(* IEC 61131-3 sources: Lasal/CPU_5344_V01/Class/SdiasManager (part 3) *)

            aProperties[1].udPropertyId     := SDM_PROP_BITMAP_APPLICATION_LED_16_31;
            aProperties[1].udPropertyValue  := AppliLEDStates[4]$UDINT;

            aProperties[2].udPropertyId     := SDM_PROP_BITMAP_APPLICATION_LED_32_47;
            aProperties[2].udPropertyValue  := AppliLEDStates[8]$UDINT;

            aProperties[3].udPropertyId     := SDM_PROP_BITMAP_APPLICATION_LED_48_63;
            aProperties[3].udPropertyValue  := AppliLEDStates[12]$UDINT;

            if SDIAS_iSetNodeProperties(hNodeHandle         := udNodeHandle
                                      , udPropertyCount     := 4
                                      , psPropertyValuePairs:= #aProperties[0]
                                      ) <> SDIAS_OK then
#ifdef HWC_LogError
              HWC_LogError(this, "@0067 (SdiasManager::CyWork) Failed to set the application LED states via OS interface!");
#endif
              ErrorInitStep := InitSSW;
              InitSSW := _PrepareError;
              ClassState := _ManagerError;
            else
              b_NewLEDStates := FALSE;
            end_if;
          end_if;
        end_if;
      elsif AsyWriteUsage = _UsedByLED then
        b_NewLEDStates := FALSE;
        AsyWriteUsage := _NotUsed;
      end_if;
    elsif (b_PostInitFinished = FALSE) & InitStartTime & ((ops.tAbsolute - InitStartTime) > (SDIAS_INIT_BLOCK_TIMEOUT + AdditionalPostInitTime)) then
      // timeout for last init if we're stuck in a step for too long (1min). otherwise the plc would not start up, which makes it hard to show the error
#ifdef HWC_LogValue1
      HWC_LogValue1(this, "@0068 (SdiasManager::CyWork) Init has been blocked for too long! Initialisation of SDIAS Manager timed out! Blocked step: 0x{0}",InitSSW$UDINT);
#endif
      ClassState := _TimeoutInInit;
      ErrorInitStep := InitSSW;
      InitSSW := _PrepareError;
    end_if;

  elsif b_PostInitFinished = FALSE then
    // if the module is not online => tell the manager that we're finished with initializing
    SendPostInitFinished(DisableThisObject:=TRUE);

    // set required error, if there is a required module
    SetRequiredError();
  end_if;

  PostRtMessages();

	state := READY;

END_FUNCTION

FUNCTION VIRTUAL GLOBAL SdiasManager::RtWork
	VAR_INPUT
		EAX 	: UDINT;
	END_VAR
	VAR_OUTPUT
		state (EAX) 	: UDINT;
	END_VAR
  VAR
  	calloption          : UDINT;
    i                   : UDINT;
    pModuleInfo         : ^t_ModuleObjectInfo;
    dataSETRUNSTATE     : t_SetRunStateCfg;
    dataResetDO         : t_ResetDOCfg;
    dataSyncData        : t_SyncData;
  	tempCmd             : CmdStruct;
    _result             : results;
    pHelpAccess         : ^t_AccessElement;
    CheckRetryCounters  : BOOL;
    ActFrameCounter     : UDINT;
    TempControlByte     : t_SDIAS_ControlByte;
    dataUPDATEDO        : t_UpdateDOCfg;
    aProperties         : ARRAY [0..4] OF SDM_PROPERTY_VALUE_PAIR;
    SyncInjectionCfg    : t_SyncInjectionCfg;
    CrashThisTime       : USINT;
    aCrashMessage       : ARRAY [0..255] OF CHAR;
    TmpRetryCount       : UDINT;
    TempUDINT           : UDINT;
    ret_code 	          : iprStates;

#ifdef SDIAS_RT_TIME_MEASUREMENT
    Time1           : UDINT;
    Time2           : UDINT;
    TimeTotal1      : UDINT;
    TimeTotal2      : UDINT;
#endif
  END_VAR

  // Called from BusInterface on UpdateRt or UpdateRtPostScan

  // Save state
  // This must be the 1. line in this function or EAX may be overwriten by the generated AWL code
  calloption := EAX;

  if Online then
    pModuleInfo := #ModuleObjInfo[0];
    case RtSSW of
//**********************************************************************************************************************************************************
      _RtIdle: // nothing

//**********************************************************************************************************************************************************
      _CreateAndModifyDOs: // create and modify ISO DOs
        CreateAndModifyIsoDOs();

        RtSSW := _Wait4DOs;

//**********************************************************************************************************************************************************
      _Wait4DOs:
        if calloption = CALL_OPTION_RT_PRESCAN then    // Called from UpdateRt
          // wait until the DOs can be activated
          if b_Ready4Rt then

            // reset data objects is only needed for connection over VARAN
            if ConnectionType = SDIAS_CON_VIA_VARAN_uC then
              // reset data objects (calculate retry timeout) - must be done every connect because at disconnect the retry time could be set with 0 byte data length
              tempCmd.uiCmd     := _BUS_IF_RESET_DO;
              tempCmd.aPara[0]  := (#dataResetDO)$DINT;

#ifndef SDIAS_DEACTIVATE_TASK_CHECKS
              dataResetDO.Handle := TaskInfoDO.Handle;

              ToBusInterface.NewInst(pPara:=#tempCmd, pResult:=#_result);

              if _result.aData[0]$t_BusIFRetvalErrorcode <> _BUS_IF_RETVAL_OK then
                // remember the log message and write it in cyclic priority to avoid a rt runtime error
                CyclicMsgMarker.PostIt.TaskInfoRunFailed := TRUE;
              end_if;
#endif

              dataResetDO.Handle := ISOReadDO.Handle;

              ToBusInterface.NewInst(pPara:=#tempCmd, pResult:=#_result);
              if _result.aData[0]$t_BusIFRetvalErrorcode <> _BUS_IF_RETVAL_OK then
                // remember the log message and write it in cyclic priority to avoid a rt runtime error
                CyclicMsgMarker.PostIt.IsoReadRunFailed := TRUE;
              end_if;

              dataResetDO.Handle := ISOWriteDO.Handle;

              ToBusInterface.NewInst(pPara:=#tempCmd, pResult:=#_result);
              if _result.aData[0]$t_BusIFRetvalErrorcode <> _BUS_IF_RETVAL_OK then
                // remember the log message and write it in cyclic priority to avoid a rt runtime error
                CyclicMsgMarker.PostIt.IsoWriteRunFailed := TRUE;
              end_if;
            end_if;

            // activate the ISO DOs

            // general settings needed for all DOs
            dataSETRUNSTATE.NewRunState := _BUS_IF_RUN_STATE_CONT_RUN;
            tempCmd.uiCmd         := _BUS_IF_SET_RUN_STATE;
            tempCmd.aPara[0]      := (#dataSETRUNSTATE)$DINT;

#ifndef SDIAS_DEACTIVATE_TASK_CHECKS

            if ConnectionType = SDIAS_CON_VIA_VARAN_uC then
              // set runstate of taskinfo read
              dataSETRUNSTATE.Handle      := TaskInfoDO.Handle;

              ToBusInterface.NewInst(pPara:=#tempCmd, pResult:=#_result);

              if _result.aData[0]$t_BusIFRetvalErrorcode <> _BUS_IF_RETVAL_OK then
                // remember the log message and write it in cyclic priority to avoid a rt runtime error
                CyclicMsgMarker.PostIt.TaskInfoRunFailed := TRUE;
              end_if;
            end_if;
#endif

            // set runstate of read
            dataSETRUNSTATE.Handle      := ISOReadDO.Handle;

            ToBusInterface.NewInst(pPara:=#tempCmd, pResult:=#_result);

            if _result.aData[0]$t_BusIFRetvalErrorcode <> _BUS_IF_RETVAL_OK then
              // remember the log message and write it in cyclic priority to avoid a rt runtime error
              CyclicMsgMarker.PostIt.IsoReadRunFailed := TRUE;
            end_if;

            // set runstate of write
            dataSETRUNSTATE.Handle      := ISOWriteDO.Handle;

            ToBusInterface.NewInst(pPara:=#tempCmd, pResult:=#_result);

            if _result.aData[0]$t_BusIFRetvalErrorcode <> _BUS_IF_RETVAL_OK then
              // remember the log message and write it in cyclic priority to avoid a rt runtime error
              CyclicMsgMarker.PostIt.IsoWriteRunFailed := TRUE;
            end_if;

            if ConnectionType = SDIAS_CON_VIA_VARAN_uC then

              // change config DO => change task config settings for Iso Read Task)
              ISOConfigWrDO.Offset := SDIAS_OFFSET_TASK_CONFIG_1;
              ISOConfigWrDO.Length := sizeof(t_TaskConfig);

              dataUPDATEDO.Handle               := ISOConfigWrDO.Handle;
              dataUPDATEDO.ud_addressoff_write  := ISOConfigWrDO.Offset;
              dataUPDATEDO.ud_length_write      := ISOConfigWrDO.Length;

              tempCmd.uiCmd         := _BUS_IF_UPDATE_DO;
              tempCmd.aPara[0]      := (#dataUPDATEDO)$DINT;

              ToBusInterface.NewInst(pPara:=#tempCmd, pResult:=#_result);

              if _result.aData[0]$t_BusIFRetvalErrorcode <> _BUS_IF_RETVAL_OK then
                // remember the log message and write it in cyclic priority to avoid a rt runtime error
                CyclicMsgMarker.PostIt.IsoConfigWrChangeFailed := TRUE;
              else
                // use the task config data
                ISOConfigWrDO.pData^$t_TaskConfig := ISOTaskConfig;
              end_if;

              dataSETRUNSTATE.NewRunState := _BUS_IF_RUN_STATE_SINGLE_RUN;
              dataSETRUNSTATE.Handle      := ISOConfigWrDO.Handle;

              tempCmd.uiCmd               := _BUS_IF_SET_RUN_STATE;
              tempCmd.aPara[0]            := (#dataSETRUNSTATE)$DINT;

              ToBusInterface.NewInst(pPara:=#tempCmd, pResult:=#_result);

              if _result.aData[0]$t_BusIFRetvalErrorcode <> _BUS_IF_RETVAL_OK then
                // remember the log message and write it in cyclic priority to avoid a rt runtime error
                CyclicMsgMarker.PostIt.IsoConfigWrTaskConfigFailed := TRUE;
              end_if;

            else
              aProperties[0].udPropertyId     := SDM_PROP_TASK_CONTROL_DURATION_TIMEOUT;
              aProperties[0].udPropertyValue  := ISOTaskConfig.TaskDurationTimeout_us;

              aProperties[1].udPropertyId     := SDM_PROP_TASK_CONTROL_CONFIGURATION;
              aProperties[1].udPropertyValue  := ISOTaskConfig.Config;

              if SDIAS_iSetNodePropertiesIndex(hNodeHandle      := udNodeHandle
                                        , udIndex               := 1
                                        , udPropertyCount       := 2
                                        , psPropertyValuePairs  := #aProperties[0]
                                        ) <> SDIAS_OK then
                CyclicMsgMarker.PostIt.IsoTaskConfigFailed := TRUE;
              end_if;

              // reconfigure PLL to ensure the SDIAS Sync refers to the correct OS tick

              // get the actual frame counter
              if SDIAS_iGetNodeProperty(hNodeHandle      :=udNodeHandle
                                      , udPropertyId     :=SDM_PROP_PLL_SYNC_TIME_FRAME_COUNTER
                                      , pudPropertyValue :=#ActFrameCounter
                                      ) = SDIAS_OK then

                tempCmd.uiCmd := _BUS_IF_SET_SYNC;

                if pPLL then
                  for i := 0 to 7 do
                    if (TaskEventIDs[i] AND 16#F0) = 16#10 then
                      // sync out is connected, take lower nibble as syncout index
                      if PLL_iGetSyncOutProperty(pPLL, ud_NodeHandlePLL, (TaskEventIDs[i] AND 16#0F), PLL_PROP_SO_SYNC_OUT_ID, #TempUDINT) = PLL_OK then
                        if TempUDINT = SDIAS_MANAGER_SYNC_SYNCOUT_ID then
                          exit;
                        end_if;
                      end_if;
                    end_if;
                  end_for;
                  dataSyncData.us_sync_nr := TaskEventIDs[i]; // iso read trigger
                else
                  dataSyncData.us_sync_nr := SDIAS_EVENT_MASK_ID_SYNC_OUT2; // iso read trigger
                end_if;

                dataSyncData.us_period_multiplier := 0;
                dataSyncData.sd_offset := 0;

                // start with the next correct sync
                dataSyncData.us_frame_count_threshold := (ActFrameCounter + 1 + (ud_BusTime_ns / 1000) / ud_SystemPeriodTime)$USINT;
                dataSyncData.us_enable_frame_count := 1;

                tempCmd.aPara[0] := (#dataSyncData)$DINT;

                ToBusInterface.NewInst(pPara:=#tempCmd, pResult:=#_result);

                if _result.aData[0]$t_BusIFRetvalErrorcode <> _BUS_IF_RETVAL_OK then
                  CyclicMsgMarker.PostIt.SetSyncFailed := TRUE;
                end_if;
              else
                CyclicMsgMarker.PostIt.GetFrameCounterFailed := TRUE;
              end_if;
            end_if;

            // stop asynchron watchdog triggering, because the watchdog gets triggered by rt now
            b_WdTriggerActive := FALSE;
            ToggleReadTaskActive := FALSE;
            b_SendWdTrigger := FALSE;

            if AsyWriteUsage = _UsedByWD then
              AsyWriteUsage := _NotUsed;
            end_if;

            PreOpCount := 0;
            RtSSW := _Wait4PllSync;
          end_if;
        end_if;

//**********************************************************************************************************************************************************
      _Wait4PllSync:
        if calloption = CALL_OPTION_RT_PRESCAN then    // Called from UpdateRt

          if PreOpCount < SDIAS_CYCLES_WAIT_AFTER_SYNC_ENABLE-1 then
            PreOpCount += 1;
          else
            PreOpCount := 0;
            RtSSW := _Wait2Ticks;
          end_if;
        end_if;

//**********************************************************************************************************************************************************
      _Wait2Ticks:  // SDIAS Manager FPGA measures the sync interval during the first to cycles
        if calloption = CALL_OPTION_RT_PRESCAN then    // Called from UpdateRt

          if PreOpCount < (SDIAS_SYNC_MEASURE_TICKS-1) then
            PreOpCount += 1;

            // we select the read task for sync, there are no sync task trigger losses allowed and we enable the sync injection
            SyncInjectionCfg := 16#03;

            if ConnectionType = SDIAS_CON_VIA_VARAN_uC then
              // change config DO => change trigger unit settings (also use trigger unit for read task)
              ISOConfigWrDO.Offset := SDIAS_OFFSET_SYNC_INJECTION_CFG;
              ISOConfigWrDO.Length := sizeof(t_SyncInjectionCfg);

              dataUPDATEDO.Handle               := ISOConfigWrDO.Handle;
              dataUPDATEDO.ud_addressoff_write  := ISOConfigWrDO.Offset;
              dataUPDATEDO.ud_length_write      := ISOConfigWrDO.Length;

              tempCmd.uiCmd         := _BUS_IF_UPDATE_DO;
              tempCmd.aPara[0]      := (#dataUPDATEDO)$DINT;

              ToBusInterface.NewInst(pPara:=#tempCmd, pResult:=#_result);

              if _result.aData[0]$t_BusIFRetvalErrorcode <> _BUS_IF_RETVAL_OK then
                // remember the log message and write it in cyclic priority to avoid a rt runtime error
                CyclicMsgMarker.PostIt.IsoConfigWrChange2Failed := TRUE;
              else
                // use the sync injection data
                ISOConfigWrDO.pData^$t_SyncInjectionCfg := SyncInjectionCfg;
              end_if;

              dataSETRUNSTATE.NewRunState := _BUS_IF_RUN_STATE_SINGLE_RUN;
              tempCmd.uiCmd               := _BUS_IF_SET_RUN_STATE;
              tempCmd.aPara[0]            := (#dataSETRUNSTATE)$DINT;

              dataSETRUNSTATE.Handle      := ISOConfigWrDO.Handle;

              ToBusInterface.NewInst(pPara:=#tempCmd, pResult:=#_result);

              if _result.aData[0]$t_BusIFRetvalErrorcode <> _BUS_IF_RETVAL_OK then
                // remember the log message and write it in cyclic priority to avoid a rt runtime error
                CyclicMsgMarker.PostIt.IsoConfigWrSyncInjFailed := TRUE;
              end_if;
            else
              aProperties[0].udPropertyId     := SDM_PROP_SYNC_INJECTION_CONFIG;
              aProperties[0].udPropertyValue  := SyncInjectionCfg;

              if SDIAS_iSetNodeProperties(hNodeHandle         := udNodeHandle
                                        , udPropertyCount     := 1
                                        , psPropertyValuePairs:= #aProperties[0]
                                        ) <> SDIAS_OK then
                // remember the log message and write it in cyclic priority to avoid a rt runtime error
                CyclicMsgMarker.PostIt.IsoSyncInjFailed := TRUE;
              end_if;
            end_if;
          else
            if ConnectionType = SDIAS_CON_VIA_VARAN_uC then
              // change config DO => change trigger unit settings (also use trigger unit for read task)
              ISOConfigWrDO.Offset := SDIAS_OFFSET_TRIGGER_UNIT_SETUP_0;
              ISOConfigWrDO.Length := sizeof(t_TriggerUnitSetup);

              dataUPDATEDO.Handle               := ISOConfigWrDO.Handle;
              dataUPDATEDO.ud_addressoff_write  := ISOConfigWrDO.Offset;
              dataUPDATEDO.ud_length_write      := ISOConfigWrDO.Length;

              tempCmd.uiCmd         := _BUS_IF_UPDATE_DO;
              tempCmd.aPara[0]      := (#dataUPDATEDO)$DINT;

              ToBusInterface.NewInst(pPara:=#tempCmd, pResult:=#_result);

              if _result.aData[0]$t_BusIFRetvalErrorcode <> _BUS_IF_RETVAL_OK then
                // remember the log message and write it in cyclic priority to avoid a rt runtime error
                CyclicMsgMarker.PostIt.IsoConfigWrChangeFailed := TRUE;
              else
                // use the trigger unit setup data
                ISOConfigWrDO.pData^$t_TriggerUnitSetup := ISOTriggerUnitSetup;
              end_if;

              dataSETRUNSTATE.NewRunState := _BUS_IF_RUN_STATE_SINGLE_RUN;
              tempCmd.uiCmd               := _BUS_IF_SET_RUN_STATE;
              tempCmd.aPara[0]            := (#dataSETRUNSTATE)$DINT;

              dataSETRUNSTATE.Handle      := ISOConfigWrDO.Handle;

              ToBusInterface.NewInst(pPara:=#tempCmd, pResult:=#_result);

              if _result.aData[0]$t_BusIFRetvalErrorcode <> _BUS_IF_RETVAL_OK then
                // remember the log message and write it in cyclic priority to avoid a rt runtime error
                CyclicMsgMarker.PostIt.IsoConfigWrTriggerUnitFailed := TRUE;
              end_if;
            else
              aProperties[0].udPropertyId     := SDM_PROP_TASK_TRIGGER_UNIT_CONTROL;
              aProperties[0].udPropertyValue  := to_udint(ISOTriggerUnitSetup.TaskSelect);

              aProperties[1].udPropertyId     := SDM_PROP_TASK_TRIGGER_UNIT_START_ADDR_RANGE;
              aProperties[1].udPropertyValue  := to_udint(ISOTriggerUnitSetup.StartAddress);

              if SDIAS_iSetNodePropertiesIndex(hNodeHandle          := udNodeHandle
                                              , udIndex             := 0
                                              , udPropertyCount     := 2
                                              , psPropertyValuePairs:= #aProperties[0]
                                              ) <> SDIAS_OK then
                CyclicMsgMarker.PostIt.IsoTriggerUnitConfigFailed := TRUE;
              end_if;
            end_if;

            // tell the manager that our sync is running, which triggers the watchdog on the modules from now on
            tempCmd.uiCmd := _BUS_IF_RT_SYNC_READY;
            ToBusInterface.NewInst(pPara:=#tempCmd, pResult:=#_result);

            // sync is starting with this RT => deactivate the watchdog trigger (no longer needed)
  #pragma warning(disable: 74)
            TempControlByte := 0;
            TempControlByte.EnableDO := FALSE;
  #pragma warning(default: 74)
            (ISOWriteDO.pData$^t_SDIAS_ControlByte + SDIAS_TRIGGER_UNIT_BYTE_SIZE)^ := TempControlByte;

            PreOpCount := 0;
            RtSSW := _PreOperational;

            if ( SupportedFeatures.TimeBroadCastSupported ) then

              uiSyncCountDown := SDIAS_SYNCSTART_COUNTDOWN;

              // Ensure that the countdown lasts at least SDIAS_SYNCSTART_COUNTDOWN ms even if the Bus time is faster than 1ms
              if ud_BusTime_ns < 1000000 then
                uiSyncCountDown *= (1000000 / ud_BusTime_ns)$UINT;
              end_if;

              //+1 because we always decrement before sending,
              // the return value of SendSyncCntDown() is the value just sent.
              uiSyncCountDown += 1;

              // Set MSB
              uiSyncCountDown := uiSyncCountDown OR 16#8000;

              // skip PreOpCount because CntDownSyn takes longer and
              // calls to UpdateRt must come directly after UpdateRtPreOp
              PreOpCount  := SDIAS_TASKINFO_READY_TICKS;
              RtSSW       := _CntDownSyncStart;
            end_if;

          end_if;
        end_if;

//**********************************************************************************************************************************************************
      _CntDownSyncStart:

        if calloption = CALL_OPTION_RT_PRESCAN then    // Called from UpdateRt

          // Call Modules so they can safe the togle bit prio the first sync
          for i := 0 to MaxPlace do
            if (pModuleInfo^.pThis) & (pModuleInfo^.pInitState) then

              if (pModuleInfo^.pInitState^ = _ClassOk) then
                pModuleInfo^.pThis^.UpdateRtPreOp(SDIAS_RTPREOP_CHECKSYNC);
              end_if;

            end_if;

            pModuleInfo += sizeof(t_ModuleObjectInfo);
          end_for;

          // Send Sync countdown
          if SendSyncCntDown() <= 16#8000 then
            udTimeMark1stSync := ops.tAbsolute;
            RtSSW := _PreOperationalWait4DataReady;
          end_if;

        end_if;

//**********************************************************************************************************************************************************
      _PreOperationalWait4DataReady:

        if calloption = CALL_OPTION_RT_PRESCAN then    // Called from UpdateRt
          SendTimeBroadCast();

          ret_code := READY;

          // Timeoutueberwachung,
          if ((ops.tAbsolute - udTimeMark1stSync) < SDIAS_PREOP_DATAVALID_TIMEOUT) then

            // Call Modules to check for dataready
            for i := 0 to MaxPlace do
              if (pModuleInfo^.pThis) & (pModuleInfo^.pInitState) then

                if (pModuleInfo^.pInitState^ = _ClassOk) then
                  if (pModuleInfo^.pThis^.UpdateRtPreOp(SDIAS_RTPREOP_CHECKDATAVALID) = BUSY) then
                    ret_code := BUSY; // Only assign if busy, check later is for any busy
                  end_if;
                end_if;

              end_if;

              pModuleInfo += sizeof(t_ModuleObjectInfo);
            end_for;

            // All Modules are done
            if (ret_code <> BUSY) then
              RtSSW := _PreOperational;
            end_if;

          else // Timeout abgelaufen

            // Call Modules to check for dataready
            for i := 0 to MaxPlace do
              if (pModuleInfo^.pThis) & (pModuleInfo^.pInitState) then

                if (pModuleInfo^.pInitState^ = _ClassOk) then
                  if (pModuleInfo^.pThis^.UpdateRtPreOp(SDIAS_RTPREOP_CHECKDATAVALID) <> READY) then
                    // Set Modul to error if it does not return READY on the last attempt.
                    pModuleInfo^.pInitState^ := _TimeoutInInit;
                  end_if;
                end_if;

              end_if;

              pModuleInfo += sizeof(t_ModuleObjectInfo);
            end_for;

            RtSSW := _PreOperational;

          end_if;
        end_if;

//**********************************************************************************************************************************************************
      _PreOperational: // we have to make 1 step between start of DOs and operational => task status bits are not valid the first time
        if calloption = CALL_OPTION_RT_PRESCAN then    // Called from UpdateRt

          SendTimeBroadCast();

          if PreOpCount < SDIAS_TASKINFO_READY_TICKS then
            PreOpCount += 1;
          else
            // finalize cyclic ssw
            if InitSSW = _WaitForRtOperational then
              ClassState  := _ClassOk;
              InitSSW     := _InitFinished;
              if ConnectionType = SDIAS_CON_VIA_VARAN_uC then
                // data is valid -> set online server to 1
                tempCmd.uiCmd    := _BUS_IF_SET_ONLINE;
                tempCmd.aPara[0] := 1;

                ToBusInterface.NewInst(pPara:=#tempCmd, pResult:=#_result);

                if _result.aData[0]$t_BusIFRetvalErrorcode <> _BUS_IF_RETVAL_OK then
                  // remember the log message and write it in cyclic priority to avoid a rt runtime error
                  CyclicMsgMarker.PostIt.SetOnlineStateFailed := TRUE;
                end_if;
              end_if;
            end_if;

            RtSSW := _Operational;

            //Set Classstates of the single modules and call the UpdateRt method to ensure valid data on the module servers if we set the state to _ClassOk.
            for i := 0 to MaxPlace do
              if pModuleInfo^.pThis then
                if pModuleInfo^.pInitState then

                  //Set ClassState of module, before calls of UpdateRt, since there are some modules which check the classstate in the UpdateRt Method
                  pModuleInfo^.pThis^.ClassState := pModuleInfo^.pInitState^;

                  if pModuleInfo^.bPreScan & (pModuleInfo^.pInitState^ = _ClassOk) then
                    // call all objects which are marked for prescan, to ensure valid data on user if classtate is class ok
                    pModuleInfo^.pThis^.UpdateRt();
                  end_if;
                else
                 //not possible
                end_if;
              end_if;
              pModuleInfo += sizeof(t_ModuleObjectInfo);
            end_for;
          end_if;

        elsif calloption = CALL_OPTION_RT_POSTSCAN then

          // dont call the postscan of modules here. It would be to early, so the DOs dont have the right state-bits.
          // The corresponding postscan-call for the UpdateRT call from this step will already be called in the "operational-case", due to the RtSSW already increased.

        end_if;
//**********************************************************************************************************************************************************
      _Operational:
        if calloption = CALL_OPTION_RT_PRESCAN then    // Called from UpdateRt

#ifdef SDIAS_RT_TIME_MEASUREMENT
          TimeTotal1 := OS_READMICROSEC();
#endif

          CrashThisTime := 0;

#ifndef SDIAS_DEACTIVATE_TASK_CHECKS

          // check if there was a retry
          CheckRetryCounters := WriteTaskInfo.pReadData^.Handshake.AnyRetries | ReadTaskInfo.pReadData^.Handshake.AnyRetries;

          // check toggle bit after first run
          if WriteTaskInfo.MaxDuration then
            if WriteTaskInfo.bOldToggle = WriteTaskInfo.pReadData^.Handshake.Toggle then
              WriteTaskInfo.ToggleErrorCount += 1;
              IsoTaskErrorCount += 1;
              CyclicMsgMarker.PostIt.ToggleErrorWrTask := TRUE;

              ClassState := _TimesliceErrorIRQ;
              Online := 0;

              DisableBus();

              if b_IsRequired then
                CrashThisTime := 1;
                _strcpy(dest:=#aCrashMessage[0], src:="Error in SDIAS write task occured! (Toggle Bit)");
              end_if;
            end_if;
          end_if;
          WriteTaskInfo.bOldToggle := WriteTaskInfo.pReadData^.Handshake.Toggle;

          // check toggle bit after first run
          if ReadTaskInfo.MaxDuration then
            if ReadTaskInfo.bOldToggle = ReadTaskInfo.pReadData^.Handshake.Toggle then
              ReadTaskInfo.ToggleErrorCount += 1;
              IsoTaskErrorCount += 1;
              CyclicMsgMarker.PostIt.ToggleErrorRdTask := TRUE;

              ClassState := _TimesliceError;
              Online := 0;

              DisableBus();

              if b_IsRequired then
                CrashThisTime := 1;
                _strcpy(dest:=#aCrashMessage[0], src:="Error in SDIAS read task occured! (Toggle Bit)");
              end_if;
            end_if;
          end_if;
          ReadTaskInfo.bOldToggle := ReadTaskInfo.pReadData^.Handshake.Toggle;

          // check executed bit always
          if (WriteTaskInfo.pReadData^.Handshake.Executed = 0) then
            WriteTaskInfo.ErrorCount += 1;
            IsoTaskErrorCount += 1;

            CyclicMsgMarker.PostIt.WrTaskNotFinished := TRUE;

            ClassState := _TimesliceErrorIRQ;
            Online := 0;

            DisableBus();

            if b_IsRequired then
              CrashThisTime := 1;
              _strcpy(dest:=#aCrashMessage[0], src:="Error in SDIAS write task occured! (Not Executed)");
            end_if;
          end_if;

          if WriteTaskInfo.pReadData^.Handshake.Error & (WriteTaskInfo.pReadData^.ErrorInfoFlags AND SDIAS_ERROR_INFO_MASK) then
            WriteTaskInfo.ErrorCount += 1;
            IsoTaskErrorCount += 1;

            CyclicMsgMarker.PostIt.ErrorWrTask := TRUE;

            ClassState := _TimesliceErrorIRQ;
            Online := 0;

            DisableBus();

            if b_IsRequired then
              CrashThisTime := 1;
              _strcpy(dest:=#aCrashMessage[0], src:="Error in SDIAS write task occured! (Error)");
            end_if;
          end_if;

          // check executed bit always
          if (ReadTaskInfo.pReadData^.Handshake.Executed = 0) & (ReadTaskInfo.pReadData^.Handshake.StatusWait = 0) then
            ReadTaskInfo.ErrorCount += 1;
            IsoTaskErrorCount += 1;

            CyclicMsgMarker.PostIt.RdTaskNotFinished := TRUE;

            ClassState := _TimesliceError;
            Online := 0;

            DisableBus();

            if b_IsRequired then
              CrashThisTime := 1;
              _strcpy(dest:=#aCrashMessage[0], src:="Error in SDIAS read task occured! (Not Executed)");
            end_if;
          end_if;

          if (ReadTaskInfo.pReadData^.Handshake.Executed = 0) & (ReadTaskInfo.pReadData^.Handshake.StatusWait = 1) then
            ReadTaskInfo.ErrorCount += 1;
            IsoTaskErrorCount += 1;

            CyclicMsgMarker.PostIt.RdTaskNoEvent := TRUE;

            ClassState := _TimesliceErrorIRQ;
            Online := 0;

            DisableBus();

            if b_IsRequired then
              CrashThisTime := 1;
              _strcpy(dest:=#aCrashMessage[0], src:="Error in SDIAS read task occured! (No Event Occured)");
            end_if;
          end_if;

          if ReadTaskInfo.pReadData^.Handshake.Error & (ReadTaskInfo.pReadData^.ErrorInfoFlags AND SDIAS_ERROR_INFO_MASK) then

            ReadTaskInfo.ErrorCount += 1;
            IsoTaskErrorCount += 1;

            CyclicMsgMarker.PostIt.ErrorRdTask := TRUE;

            ClassState := _TimesliceError;
            Online := 0;

            DisableBus();

            if b_IsRequired then
              CrashThisTime := 1;
              _strcpy(dest:=#aCrashMessage[0], src:="Error in SDIAS read task occured! (Error)");
            end_if;
          end_if;

          //Check if SdiasManager FPGA supports the detection of TimeSliceErrorIRQ
          if FeatureInfo.OptionBits.TaskInterruptionDetectionSupported = TRUE then
            //Check if error info flag bit 0 is set .. SYNC occured while Task was executing
            if WriteTaskInfo.pReadData^.ErrorInfoFlags.AccessCanceled = TRUE then
              WriteTaskInfo.ErrorCount += 1;
              IsoTaskErrorCount += 1;

              CyclicMsgMarker.PostIt.WrTaskInterruptedByRdTask := TRUE;

              ClassState := _TimesliceErrorIRQ;
              Online := 0;

              DisableBus();

              if b_IsRequired then
                CrashThisTime := 1;
                _strcpy(dest:=#aCrashMessage[0], src:="Error in SDIAS write task occured! (Interrupted by RdTask)");
              end_if;
            end_if;
          end_if;

          // show the task duration on the servers and remember the max duration
          IsoWrTaskDuration := WriteTaskInfo.pReadData^.DurationTime;
          if IsoWrTaskDuration > WriteTaskInfo.MaxDuration then
            WriteTaskInfo.MaxDuration := IsoWrTaskDuration;
          end_if;

          //own if because user can reset the server
          if IsoWrTaskDuration > IsoWrTaskMaxDuration then
            IsoWrTaskMaxDuration := IsoWrTaskDuration;
          end_if;

          // show the task duration on the servers and remember the max duration
          IsoRdTaskDuration := ReadTaskInfo.pReadData^.DurationTime;
          if IsoRdTaskDuration > ReadTaskInfo.MaxDuration then
            ReadTaskInfo.MaxDuration := IsoRdTaskDuration;
          end_if;

          //own if because user can reset the server
          if IsoRdTaskDuration > IsoRdTaskMaxDuration then
            IsoRdTaskMaxDuration := IsoRdTaskDuration;
          end_if;

#else
#pragma message("ATTENTION: TASK CHECKS FOR SDIAS ARE DEACTIVATED!")

#ifdef SDIAS_CHECK_ALL_RETRIES
          CheckRetryCounters := TRUE;
#else
          CheckRetryCounters := FALSE;
#pragma message("ATTENTION: RETRY CHECKS FOR SDIAS ARE DEACTIVATED!")
#endif
#endif

          SendTimeBroadCast();

          // check accesses for errors
          for i := 0 to MaxPlace do
            // if the state is ok
            if pModuleInfo^.bPreScan & (pModuleInfo^.pThis^.ClassState = _ClassOk) then
              if CheckRetryCounters then
                TmpRetryCount := 0;
                // check default accesses for error
                if pModuleInfo^.pDefaultAccesses^.ReadAccess.pStateByte then
                  // increase retrycounter if retries occured on the access
                  TmpRetryCount += CheckAccess(bsStateByte    := pModuleInfo^.pDefaultAccesses^.ReadAccess.pStateByte^
                                             , sdRequired     := pModuleInfo^.Required
                                             , sdPlace        := i$DINT
                                             , pCrashThisTime := #CrashThisTime
                                             , pCrashMessage  := #aCrashMessage[0]
                                             );
                end_if;

                if pModuleInfo^.pDefaultAccesses^.WriteAccess.pStateByte then
                  // increase retrycounter if retries occured on the access
                  TmpRetryCount += CheckAccess(bsStateByte    := pModuleInfo^.pDefaultAccesses^.WriteAccess.pStateByte^
                                             , sdRequired     := pModuleInfo^.Required
                                             , sdPlace        := i$DINT
                                             , pCrashThisTime := #CrashThisTime
                                             , pCrashMessage  := #aCrashMessage[0]
                                             );
                end_if;

                // check all special accesses for errors
                pHelpAccess := pModuleInfo^.pFirstAccess;
                while pHelpAccess do
                  // increase retrycounter if retries occured on the access
                  TmpRetryCount += CheckAccess(bsStateByte    := pHelpAccess^.ppStateByte^^
                                             , sdRequired     := pModuleInfo^.Required
                                             , sdPlace        := i$DINT
                                             , pCrashThisTime := #CrashThisTime
                                             , pCrashMessage  := #aCrashMessage[0]
                                             );

                  pHelpAccess := pHelpAccess^.pNext;
                end_while;

                // update retrycounter
                pModuleInfo^.pThis^.RetryCounter += TmpRetryCount;
                RetryCounter += TmpRetryCount;

              end_if;
#ifdef SDIAS_RT_TIME_MEASUREMENT
              Time1 := OS_READMICROSEC();
#endif

              // call them only if we're not about to crash
              if CrashThisTime = 0 then
                // call all objects which are marked for prescan
                pModuleInfo^.pThis^.UpdateRt();
              end_if;

#ifdef SDIAS_RT_TIME_MEASUREMENT
              Time2 := OS_READMICROSEC();
              pModuleInfo^.RtTime_us := Time2 - Time1;
              if pModuleInfo^.RtTime_us > pModuleInfo^.RtTimeMax_us then
                pModuleInfo^.RtTimeMax_us := pModuleInfo^.RtTime_us;
              end_if;
#endif
            end_if;
            pModuleInfo += sizeof(t_ModuleObjectInfo);
          end_for;

          if CrashThisTime then
            // print pending error messages before crash
            PostRtMessages();

            if CrashThisTime = 1 then
              SDIAS_iReportEvent(uiEvent:=SDM_EVENT_ERROR_REQUIRED_MODULE, pucEvntMsg:=#aCrashMessage[0]);

            elsif CrashThisTime = 2 then
              // set required error (don't use SetRequiredError method, because logging in realtime could cause a rt runtime error which will disguise our required error)
              tempCmd.uiCmd     := _BUS_IF_SET_REQUIRED_ERROR;

              ToBusInterface.NewInst(pPara:=#tempCmd, pResult:=#_result);
              if _result.aData[0]$t_BusIFRetvalErrorcode <> _BUS_IF_RETVAL_OK then
                CyclicMsgMarker.PostIt.ForwardRequiredErrorFailed := TRUE;
              end_if;
            end_if;
          end_if;

#ifdef SDIAS_RT_TIME_MEASUREMENT
          TimeTotal2 := OS_READMICROSEC();
          RtPreDuration := TimeTotal2 - TimeTotal1;
#endif

        elsif calloption = CALL_OPTION_RT_POSTSCAN then // Called from UpdateRtPostScan
#ifdef SDIAS_RT_TIME_MEASUREMENT
          TimeTotal1 := OS_READMICROSEC();
#endif

          for i := 0 to MaxPlace do
            if pModuleInfo^.bPostScan & (pModuleInfo^.pThis^.ClassState = _ClassOk) then

#ifdef SDIAS_RT_TIME_MEASUREMENT
              Time1 := OS_READMICROSEC();
#endif

              // call all objects which are marked for postscan
              pModuleInfo^.pThis^.UpdateRtPostScan();

#ifdef SDIAS_RT_TIME_MEASUREMENT
              Time2 := OS_READMICROSEC();
              pModuleInfo^.RtPostTime_us := Time2 - Time1;
              if pModuleInfo^.RtPostTime_us > pModuleInfo^.RtPostTimeMax_us then
                pModuleInfo^.RtPostTimeMax_us := pModuleInfo^.RtPostTime_us;
              end_if;
#endif

            end_if;
            pModuleInfo += sizeof(t_ModuleObjectInfo);
          end_for;

#ifdef SDIAS_RT_TIME_MEASUREMENT
          TimeTotal2 := OS_READMICROSEC();
          RtPostDuration := TimeTotal2 - TimeTotal1;
#endif
        end_if;

//**********************************************************************************************************************************************************
    end_case;
  end_if;

	state := READY;

END_FUNCTION

FUNCTION VIRTUAL GLOBAL SdiasManager::ClassState::NewInst
	VAR_INPUT
		pPara 	: ^CmdStruct;
		pResult 	: ^results;
	END_VAR
	VAR_OUTPUT
		ret_code 	: iprStates;
	END_VAR
  VAR
  	ByteNr      : USINT;
    PosInByte   : USINT;
    pDataADDMove: ^t_AddMoveDOCfg;
    Place       : UDINT;
    pAccessInfo : ^t_AccessInfoRet;
//    DAPara      : t_RDWRDOCfg;
  	tempCmd     : CmdStruct;
    _result     : results;
    sRDDADOCfg  :   t_RDWRDOCfg;

    pStr_HWTRequested     : ^CHAR;
    tmpplace      : USINT;
    pStr_HWTreeEntry : ^CHAR;
    usNextPlace   : USINT;
    i             : USINT;
  END_VAR

	ret_code := READY;

	CASE pPara^.uiCmd OF
//*****************************************************************************
//** EXTERNAL COMMANDS (FOR DIAGNOSIS)                                       **
//*****************************************************************************

//**********************************************************************************************************************************************************
    SDIAS_CMD_GET_MIB_ADDR :
      // return the address of the ManagerInfoBlock variable
      if ClassState = _ClassOk then
        pResult^.uiLng := 4;
        pResult^.aData[0]$^void := #ManagerInfoBlock$^void;
      else

        ret_code := ERROR;

        // Read the info block via DAs if we are conncted via Varan and the Classstate is _ModuleFoundButManagerIsOff
        if ConnectionType = SDIAS_CON_VIA_VARAN_uC then

          // Check Class State
          tempCmd.uiCmd := _BUS_IF_GET_CLASS_STATE;
          ret_code := ToBusInterface.NewInst(pPara:=#tempCmd, pResult:=#_result);

          if ((ret_code = READY) & (_result.aData[0]$t_BusIFRetvalErrorcode = _BUS_IF_RETVAL_OK)) then

            if (_result.aData[4]$t_e_VaranErrors = _ModuleFoundButManagerIsOff) then
              // Manager is off so we can read the ManagerInfoBlock with DA without interrupting regular bus transfer
              tempCmd.uiCmd := _BUS_IF_RD_DA;

              // prepare fetching the infoblock
              ModuleSizeNeeded :=sizeof(ManagerInfoBlock.ModuleInfos);

              sRDDADOCfg.ud_length    := 128;
              sRDDADOCfg.ud_AddOffset := 0;
              sRDDADOCfg.p_ud_data    := #ManagerInfoBlock + AccessProgress;

              tempCmd.aPara[0]$^t_RDWRDOCfg := #sRDDADOCfg;

              while ModuleSizeNeeded >= 128 do

                ret_code := ToBusInterface.NewInst(pPara:=#tempCmd, pResult:=#_result);
                if ((ret_code <> READY) & (_result.aData[0]$t_BusIFRetvalErrorcode <> _BUS_IF_RETVAL_OK)) then
                  ret_code := ERROR;
                  return;
                end_if;

                sRDDADOCfg.ud_AddOffset += 128;
                sRDDADOCfg.p_ud_data    += 128;

                ModuleSizeNeeded  -= 128;
              end_while;

              if ModuleSizeNeeded then

                sRDDADOCfg.ud_length    := ModuleSizeNeeded;

                ret_code := ToBusInterface.NewInst(pPara:=#tempCmd, pResult:=#_result);
                if ((ret_code <> READY) & (_result.aData[0]$t_BusIFRetvalErrorcode <> _BUS_IF_RETVAL_OK)) then
                  ret_code := ERROR;
                  return;
                end_if;
              end_if;

              pResult^.uiLng := 4;
              pResult^.aData[0]$^void := #ManagerInfoBlock$^void;

            else
              ret_code := ERROR;
            end_if;

          else
            ret_code := ERROR;
          end_if;
        end_if;
      end_if;

//**********************************************************************************************************************************************************
    SDIAS_CMD_GET_MOI_ADDR :
      // return the address of the ModuleObjInfo variable
      pResult^.uiLng := 4;
      pResult^.aData[0]$^void := #ModuleObjInfo$^void;

//**********************************************************************************************************************************************************
    CMD_GET_HARDWARE_DIAGNOSIS:
      //Returns module info
      ret_code := ERROR;
      pResult^.aData[0]$t_HWCGetHardwareDiagnosisOut.retcode := _HWC_RETVAL_ERROR;

      pStr_HWTRequested := pPara^.aPara[0]$t_HWCGetHardwareDiagnosisIn.pStr_HardewareTreeEntry;

      if pStr_HWTRequested &
         ( ((pStr_HWTRequested  + pPara^.aPara[0]$t_HWCGetHardwareTreeEntryIn.us_current_index  - 1)^$USINT) = HWT_ESCAPE_SDIAS ) then

        tmpplace := (pStr_HWTRequested+pPara^.aPara[0]$t_HWCGetHardwareDiagnosisIn.us_current_index)^$USINT;

        //Check if pointer is valid
        if ModuleObjInfo[tmpplace].pThis then
          ret_code := ModuleObjInfo[tmpplace].pThis^.NewInst(pPara,pResult);
        else
          pResult^.aData[0]$t_HWCGetHardwareDiagnosisOut.retcode := _HWC_RETVAL_ERROR_SDIAS_MODULE_NOT_FOUND;
        end_if;
      end_if;

//**********************************************************************************************************************************************************
    CMD_GET_HARDWARE_TREE_ENTRY:
      //Returns module info
      ret_code := ERROR;
      pResult^.aData[0]$t_HWCGetHardwareTreeEntryOut.retcode := _HWC_RETVAL_ERROR;

      pStr_HWTreeEntry := pPara^.aPara[0]$t_HWCGetHardwareTreeEntryIn.pStr_LastHardewareTreeEntry;

      //First HWT Path
      if pStr_HWTreeEntry = nil then
        if ModuleObjInfo[0].pThis then

          ret_code := ModuleObjInfo[0].pThis^.NewInst(pPara,pResult);
        else
          pResult^.aData[0]$t_HWCGetHardwareTreeEntryOut.retcode := _HWC_RETVAL_ERROR_SDIAS_MODULE_NOT_FOUND;
        end_if;

      //search next module
      elsif ( ((pStr_HWTreeEntry  + pPara^.aPara[0]$t_HWCGetHardwareTreeEntryIn.us_current_index  - 1)^$USINT) = HWT_ESCAPE_SDIAS ) then

        // Check last modul again incase it was an extension module
        usNextPlace := (pStr_HWTreeEntry  + pPara^.aPara[0]$t_HWCGetHardwareTreeEntryIn.us_current_index)^$USINT;
        if ModuleObjInfo[usNextPlace].pThis then

          ret_code := ModuleObjInfo[usNextPlace].pThis^.NewInst(pPara,pResult);
        else
          ret_code := READY;
          pResult^.aData$t_HWCGetHardwareTreeEntryOut.retcode := _HWC_RETVAL_OK_END_OF_LIST;
          return;
        end_if;

        // Module was found, return next one
        if ret_code = READY &
           (pResult^.aData$t_HWCGetHardwareTreeEntryOut.retcode = _HWC_RETVAL_OK_MODULE_FOUND |
            pResult^.aData$t_HWCGetHardwareTreeEntryOut.retcode = _HWC_RETVAL_OK_END_OF_LIST) then

          usNextPlace += 1;
          if ModuleObjInfo[usNextPlace].pThis then

            ret_code := ModuleObjInfo[usNextPlace].pThis^.NewInst(pPara,pResult);
          else
            ret_code := READY;
            pResult^.aData$t_HWCGetHardwareTreeEntryOut.retcode := _HWC_RETVAL_OK_END_OF_LIST;
          end_if;

        end_if;

      end_if;

//**********************************************************************************************************************************************************

//*****************************************************************************
//** COMMANDS FROM SDIAS MODULES                                             **
//*****************************************************************************

    // port number is always stored in pPara^.aPara[MAXCMDPARA-1]
//**********************************************************************************************************************************************************
		SDIAS_CMD_ADD_RD_ACCESS:
      if AddAccess(_Read, pPara^.aPara[0]$^SdiasBase, pPara^.aPara[1]$UDINT, pPara^.aPara[2], pPara^.aPara[3]$HINT, pPara^.aPara[4]$UINT, pPara^.aPara[5]$pVoid, pPara^.aPara[6]$pVoid, pPara^.aPara[7]$pVoid, pPara^.aPara[8]$^UDINT, pPara^.aPara[9]$UDINT, pPara^.aPara[10]$BOOL) = FALSE then
        ret_code := ERROR;
      end_if;

//**********************************************************************************************************************************************************
    SDIAS_CMD_ADD_WR_ACCESS:
      if AddAccess(_Write, pPara^.aPara[0]$^SdiasBase, pPara^.aPara[1]$UDINT, pPara^.aPara[2], pPara^.aPara[3]$HINT, pPara^.aPara[4]$UINT, pPara^.aPara[5]$pVoid, pPara^.aPara[6]$pVoid, pPara^.aPara[7]$pVoid, pPara^.aPara[8]$^UDINT, pPara^.aPara[9]$UDINT, pPara^.aPara[10]$BOOL) = FALSE then
        ret_code := ERROR;
      end_if;

//**********************************************************************************************************************************************************
		SDIAS_CMD_ADD_DYN_RD_ACCESS:
      if AddAccess(_ReadDynamic, pPara^.aPara[0]$^SdiasBase, pPara^.aPara[1]$UDINT, pPara^.aPara[2], pPara^.aPara[3]$HINT, pPara^.aPara[4]$UINT, pPara^.aPara[5]$pVoid, pPara^.aPara[6]$pVoid, pPara^.aPara[7]$pVoid, pPara^.aPara[8]$^UDINT, pPara^.aPara[9]$UDINT, pPara^.aPara[10]$BOOL) = FALSE then
        ret_code := ERROR;
      end_if;

//**********************************************************************************************************************************************************
    SDIAS_CMD_ADD_DYN_WR_ACCESS:
      if AddAccess(_WriteDynamic, pPara^.aPara[0]$^SdiasBase, pPara^.aPara[1]$UDINT, pPara^.aPara[2], pPara^.aPara[3]$HINT, pPara^.aPara[4]$UINT, pPara^.aPara[5]$pVoid, pPara^.aPara[6]$pVoid, pPara^.aPara[7]$pVoid, pPara^.aPara[8]$^UDINT, pPara^.aPara[9]$UDINT, pPara^.aPara[10]$BOOL) = FALSE then
        ret_code := ERROR;
      end_if;

//**********************************************************************************************************************************************************
    SDIAS_CMD_CHANGE_DYN_ACCESS:
      if ChangeDynAccess(AccessHandle:=pPara^.aPara[0]$UDINT, NewOffset:=pPara^.aPara[1]$UDINT, NewLength:=pPara^.aPara[2]$UDINT) = FALSE then
        ret_code := ERROR;
      end_if;

//**********************************************************************************************************************************************************
    SDIAS_CMD_SDO_SEND_REQUEST:

      if pPara^.aPara[1]$t_SDIAS_SDO_Cmd = SDIAS_SDO_CMD_SPI_READ & FirmwareVersion < SDIAS_SDO_SPI_FIRMWARE_VERSION_AVAILABLE then
#ifdef HWC_LogError
        HWC_LogError(this, "@0069 (SdiasManager::ClassState::NewInst) SPI Read failed, Update FirmwareVersion of SDIAS Manager");
#endif
        ret_code := ERROR;
        return;
      end_if;

      if AddSDOReq(pCmdSvr:=pPara^.aPara[0]$^SvrChCmd, Command:=pPara^.aPara[1]$t_SDIAS_SDO_Cmd, Place:=pPara^.aPara[2]$USINT, CmdLength:=pPara^.aPara[3]$USINT, pReqBuf:=pPara^.aPara[4]$^USINT) <> SDIAS_OK then
        ret_code := ERROR;
      end_if;

//**********************************************************************************************************************************************************
    SDIAS_CMD_CHANGE_LED_STATE:
      // get byte position ouf of place (place 0-3 in byte 0, 4-7 in byte 1,...)
      ByteNr := pPara^.aPara[1]$USINT SHR 2;
      PosInByte := (pPara^.aPara[1]$USINT AND 2#11) SHL 1;
      AppliLEDStates[ByteNr] := (AppliLEDStates[ByteNr] AND NOT(2#11 SHL PosInByte)) OR (pPara^.aPara[2]$USINT SHL PosInByte);
      b_NewLEDStates := TRUE;

//**********************************************************************************************************************************************************
    SDIAS_CMD_DA_RD_ACCESS:
      // not implemented yet
      ret_code := ERROR;

//      DaWriteBuffer.ReadLength  := pPara^.aPara[1]$USINT;
//      DaWriteBuffer.ReadOffset  := pPara^.aPara[0]$HINT;
//      DaWriteBuffer.WriteLength := 0;
//      DaWriteBuffer.WriteOffset := 0;
//
//      DaWriteBuffer.TriggerUnit := sizeof(t_DAWrPayloadFrame) - sizeof(t_DAWrPayloadFrame.Data); // no data sent on reading
//
//      DAPara.ud_AddOffset := DaWriteOffset;
//      DAPara.ud_length    := DaWriteBuffer.TriggerUnit;
//      DAPara.p_ud_data    := (#DaWriteBuffer)$^UDINT;
//
//      tempCmd.uiCmd := _BUS_IF_WR_DA;
//      tempCmd.aPara[0] := (#DAPara)$DINT;
//      ToBusInterface.NewInst(pPara:=#tempCmd, pResult:=#_result);
//
//      if _result.aData[4]$t_BusIFRetvalErrorcode <> _BUS_IF_RETVAL_OK then
//        LogError("@006A (SdiasManager::ClassState::NewInst) Direct access write on VARAN failed as part of the SDIAS direct access read!");
//        ret_code := ERROR;
//      else
//        DAPara.ud_AddOffset := DaReadOffset;
//        DAPara.ud_length    := DaWriteBuffer.ReadLength + sizeof(t_SDIAS_StateByte);
//        DAPara.p_ud_data    := (#DaReadBuffer)$^UDINT;
//
//        tempCmd.uiCmd := _BUS_IF_RD_DA;
//        tempCmd.aPara[0] := (#DAPara)$DINT;
//        ToBusInterface.NewInst(pPara:=#tempCmd, pResult:=#_result);
//
//        if _result.aData[4]$t_BusIFRetvalErrorcode <> _BUS_IF_RETVAL_OK then
//          LogError("@006B (SdiasManager::ClassState::NewInst) Direct access read on VARAN failed as part of the SDIAS direct access read!");
//          ret_code := ERROR;
//        else
//          // copy the read data to the user memory
//          _memcpy(ptr1:=pPara^.aPara[2]$^USINT, ptr2:=#DaReadBuffer.Data, cntr:=DaWriteBuffer.ReadLength);
//        end_if;
//      end_if;

//**********************************************************************************************************************************************************
    SDIAS_CMD_DA_WR_ACCESS:
      // not implemented yet
      ret_code := ERROR;

//      DaWriteBuffer.ReadLength  := 0;
//      DaWriteBuffer.ReadOffset  := 0;
//      DaWriteBuffer.WriteLength := pPara^.aPara[1]$USINT;
//      DaWriteBuffer.WriteOffset := pPara^.aPara[0]$HINT;
//
//      DaWriteBuffer.TriggerUnit := sizeof(t_DAWrPayloadFrame) - sizeof(t_DAWrPayloadFrame.Data) + DaWriteBuffer.WriteLength; // no data sent on reading
//
//      // copy the write data from the user memory
//      _memcpy(ptr1:=#DaWriteBuffer.Data, ptr2:=pPara^.aPara[2]$^USINT, cntr:=DaWriteBuffer.WriteLength);
//
//      DAPara.ud_AddOffset := DaWriteOffset;
//      DAPara.ud_length    := DaWriteBuffer.TriggerUnit;
//      DAPara.p_ud_data    := (#DaWriteBuffer)$^UDINT;
//
//      tempCmd.uiCmd := _BUS_IF_WR_DA;
//      tempCmd.aPara[0] := (#DAPara)$DINT;
//      ToBusInterface.NewInst(pPara:=#tempCmd, pResult:=#_result);
//
//      if _result.aData[4]$t_BusIFRetvalErrorcode <> _BUS_IF_RETVAL_OK then
//        LogError("@006C (SdiasManager::ClassState::NewInst) Direct access write on VARAN failed as part of the SDIAS direct access write!");
//        ret_code := ERROR;
//      else
//        DAPara.ud_AddOffset := DaReadOffset;
//        DAPara.ud_length    := sizeof(t_SDIAS_StateByte);
//        DAPara.p_ud_data    := (#DaReadBuffer)$^UDINT;
//
//        tempCmd.uiCmd := _BUS_IF_RD_DA;
//        tempCmd.aPara[0] := (#DAPara)$DINT;
//        ToBusInterface.NewInst(pPara:=#tempCmd, pResult:=#_result);
//
//        if _result.aData[4]$t_BusIFRetvalErrorcode <> _BUS_IF_RETVAL_OK then
//          LogError("@006D (SdiasManager::ClassState::NewInst) Direct access read on VARAN failed as part of the SDIAS direct access write!");
//          ret_code := ERROR;
//        end_if;
//      end_if;

//**********************************************************************************************************************************************************
    SDIAS_CMD_REQUIRED_ERROR:
      SetRequiredError(pTargetThis:=pPara^.aPara[0]$^SdiasBase, Place:=pPara^.aPara[1]$UDINT);

//**********************************************************************************************************************************************************
    SDIAS_CMD_INIT_STATE_LOGIN:
      Place := pPara^.aPara[1]$UDINT;
      if (Place <= SDIAS_MAX_PLACE_NR) & pPara^.aPara[0] then
        ModuleObjInfo[Place].pInitState       := pPara^.aPara[0]$^t_e_VaranErrors;
        ModuleObjInfo[Place].pThis            := pPara^.aPara[2]$^SdiasBase;

        // get task settings
        ModuleObjInfo[Place].bPreScan         := (pPara^.aPara[3] AND SDIAS_TASK_MASK_RT_PRE ) <> 0;
        ModuleObjInfo[Place].bPostScan        := (pPara^.aPara[3] AND SDIAS_TASK_MASK_RT_POST) <> 0;
        ModuleObjInfo[Place].bCyclic          := (pPara^.aPara[3] AND SDIAS_TASK_MASK_CY     ) <> 0;

        // get access structure
        ModuleObjInfo[Place].pDefaultAccesses := pPara^.aPara[4]$^t_SDIAS_DefaultAccesses;

        // required info
        ModuleObjInfo[Place].Required         := pPara^.aPara[5];

        if ModuleObjInfo[Place].Required & (b_SDIASModulesRequired = FALSE) then
          b_SDIASModulesRequired := TRUE;
          // if any access is required => the businterface is also required
          tempCmd.uiCmd := _BUS_IF_SET_REQUIRED;
          ToBusInterface.NewInst(pPara:=#tempCmd, pResult:=#_result);
          if _result.aData[0]$t_BusIFRetvalErrorcode <> _BUS_IF_RETVAL_OK then
#ifdef HWC_LogError
            HWC_LogError(this, "@006E (SdiasManager::ClassState::NewInst) Failed to set the BusInterface to required");
#endif
          end_if;
        end_if;

        // remember the highest place to save time in module scanning operations like calling the realtime methods
        if (Place > MaxPlace) | (MaxPlace = SDIAS_PLACE_NO_MODULE_ADDED_SO_FAR) then
          MaxPlace := Place;
        end_if;
      else
        ret_code := ERROR;
      end_if;

//**********************************************************************************************************************************************************
    SDIAS_CMD_GET_HW_PATH:
      // forward it to bus interface
      pPara^.uiCmd := _BUS_IF_GET_HW_PATH;
      ret_code := ToBusInterface.NewInst(pPara, pResult);

//**********************************************************************************************************************************************************
    SDIAS_CMD_INSTALL_CYCLIC_TASK:
      ModuleObjInfo[pPara^.aPara[0]].bCyclic := TRUE;

//**********************************************************************************************************************************************************
    SDIAS_CMD_GET_CONNECTION_TYPE:
      pResult^.uiLng := sizeof(t_SDIAS_ConnectionType);
      pResult^.aData[0]$t_SDIAS_ConnectionType := ConnectionType;

//**********************************************************************************************************************************************************
    SDIAS_CMD_CREATE_MUTEX:
      // forward it to bus interface
      pPara^.uiCmd := _BUS_IF_CREATE_MUTEX;
      ret_code := ToBusInterface.NewInst(pPara, pResult);

//**********************************************************************************************************************************************************
    SDIAS_CMD_IS_VARAN_AVAILABLE:
      // forward it to bus interface
      pPara^.uiCmd := _BUS_IF_IS_VARAN_AVAILABLE;
      ret_code := ToBusInterface.NewInst(pPara, pResult);

//**********************************************************************************************************************************************************
    SDIAS_CMD_ADD_DEVICE_ID:
    //add valid ids to list
    for i:= 0 to 9 do
      //Check if no id is stored or if id is already stored in list.
      if aValidDeviceIDs[i] = 0 | aValidDeviceIDs[i] = pPara^.aPara[0]$UDINT then
        aValidDeviceIDs[i] := pPara^.aPara[0]$UDINT;
        exit;
      end_if;
    end_for;

//**********************************************************************************************************************************************************
    SDIAS_CMD_GET_SUPPORTED_FEATURES:

      //Set length to be flexible for future
      pResult^.uiLng := 4;
      pResult^.aData[0]$BDINT := SupportedFeatures;

//**********************************************************************************************************************************************************
    CMD_EXTEND_POST_INIT_TIME:

      // use it also for ourself
      AdditionalPostInitTime += pPara^.aPara[0]$UDINT;

      // forward it to bus interface
      ret_code := ToBusInterface.NewInst(pPara, pResult);

//**********************************************************************************************************************************************************

//*****************************************************************************
//** COMMANDS FORWARDED BY SDIAS BUS INTERFACE                               **
//*****************************************************************************

//**********************************************************************************************************************************************************
    _BUS_IF_ADD_MOVE_DO:
      // correct the parameters, because the calling class doesn't have the information
      pDataADDMove                        := (pPara^.aPara[0])$^t_AddMoveDOCfg;

      pDataADDMove^.ud_handle_source      := ISOReadDO.AccessHandle;

      // if the module has no source at this time, don't calculate any addresses with the NIL pointer
      if pDataADDMove^.p_sourcedata then
        pDataADDMove^.ud_addressoff_source  := pDataADDMove^.p_sourcedata$UDINT - ISOReadDO.pData$UDINT;

        // if we have the DPRAM address extra => recalculate the address
        if ISOReadDO.pDataDPRAM then
          pDataADDMove^.p_sourcedata := ISOReadDO.pDataDPRAM + pDataADDMove^.ud_addressoff_source;
        end_if;
      end_if;

      pDataADDMove^.ud_handle_dest        := ISOWriteDO.AccessHandle;
      pDataADDMove^.ud_addressoff_dest    := pDataADDMove^.p_destdata$UDINT - ISOWriteDO.pData$UDINT;

      // if we have the DPRAM address extra => recalculate the address
      if ISOWriteDO.pDataDPRAM then
        pDataADDMove^.p_destdata := ISOWriteDO.pDataDPRAM + pDataADDMove^.ud_addressoff_dest;
      end_if;

      // forward it to bus interface
      ret_code := ToBusInterface.NewInst(pPara, pResult);

//**********************************************************************************************************************************************************
    _BUS_IF_UPDATE_MOVE_DO:
      // forward it to bus interface
      ret_code := ToBusInterface.NewInst(pPara, pResult);

//**********************************************************************************************************************************************************
    _BUS_IF_GET_ACCESS_INFO:
      // return the access info
      pResult^.uiLng := sizeof(t_AccessInfoRet);
      pAccessInfo := (#pResult^.aData[0])$^t_AccessInfoRet;

      // check if we got a valid pointer (local memory)
      if pPara^.aPara[0] then

        pAccessInfo^.ud_handle     := ISOReadDO.AccessHandle;
        pAccessInfo^.ud_addressoff := pPara^.aPara[0]$UDINT - ISOReadDO.pData$UDINT;

        // if we have the DPRAM address extra => recalculate the address
        if ISOReadDO.pDataDPRAM then
          pAccessInfo^.p_dataDPRAM := ISOReadDO.pDataDPRAM + pAccessInfo^.ud_addressoff;
        end_if;

        pAccessInfo^.retcode := _BUS_IF_RETVAL_OK;
      else
        pAccessInfo^.retcode := _BUS_IF_RETVAL_ERROR_INVALID_POINTER;
      end_if;

//**********************************************************************************************************************************************************

//*****************************************************************************
//** COMMANDS FROM BUS INTERFACE                                             **
//*****************************************************************************

//**********************************************************************************************************************************************************
    _BUS_IF_HWCONNECT :
      // device has been connected. if there is no bus ready signal or we're in the init (no bus ready in init if module is already connected) => do the connect-stuff here
      ConnectEvent();
      pResult^.aData[0] := _BUS_IF_RETVAL_OK;

//**********************************************************************************************************************************************************
    _BUS_IF_HWSUB_BUS_READY :
      // we wait for the device bitmap to match => do nothing here
      pResult^.aData[0] := _BUS_IF_RETVAL_OK;

//**********************************************************************************************************************************************************
    _BUS_IF_HWDISCONNECT :
      // device has been disconnected
      DisconnectEvent();
      pResult^.aData[0] := _BUS_IF_RETVAL_OK;

//**********************************************************************************************************************************************************
    _BUS_IF_HWINTERRUPT :
      // error at device which may lead to a disconnect or replace the disconnect callback
      InterruptEvent();
      pResult^.aData[0] := _BUS_IF_RETVAL_OK;

//**********************************************************************************************************************************************************
    _BUS_IF_CHECK_DEVICE_ID :
      // check for correct device id

      pResult^.aData[0] := (DeviceID = pPara^.aPara[0]$UDINT);
      if pResult^.aData[0] = false then
        for i:= 0 to 9 do
          //Id found?
          if aValidDeviceIDs[i] = pPara^.aPara[0]$UDINT then
            pResult^.aData[0] := TRUE;
            exit;
          end_if;
        end_for;
      end_if;

//**********************************************************************************************************************************************************
    _BUS_IF_GET_TASK_INFO:
      // we must fetch the task info before the image with the payload is copied to ensure correct data and correct error detection

      // on local SDIAS we have to fetch it from the OS
      if ConnectionType = SDIAS_CON_LOCAL_uC then
        if SDIAS_iGetNodePropertyIndexLen(hNodeHandle   := udNodeHandle
                                     , udIndex          := 1
                                     , udPropertyId     := SDM_PROP_TASK_INFO
                                     , udBufferLength   := sizeof(t_TaskInfoData) - sizeof(t_TaskInfoData.ErrorInfoFlags) - sizeof(t_TaskInfoData.Reserved)
                                     , pucBuf           := (#RdTaskInfo.Handshake)$^USINT
                                     ) <> SDIAS_OK then
          CyclicMsgMarker.PostIt.GetRdInfoFailed := TRUE;
        end_if;
        if SDIAS_iGetNodePropertyIndex(hNodeHandle      := udNodeHandle
                                     , udIndex          := 1
                                     , udPropertyId     := SDM_PROP_TASK_ERROR_INFO_FLAGS
                                     , pudPropertyValue := (#RdTaskInfo.ErrorInfoFlags)$^UDINT
                                     ) <> SDIAS_OK then
          CyclicMsgMarker.PostIt.GetRdInfoFailed := TRUE;
        end_if;

        if SDIAS_iGetNodePropertyIndexLen(hNodeHandle   := udNodeHandle
                                     , udIndex          := 2
                                     , udPropertyId     := SDM_PROP_TASK_INFO
                                     , udBufferLength   := sizeof(t_TaskInfoData) - sizeof(t_TaskInfoData.ErrorInfoFlags) - sizeof(t_TaskInfoData.Reserved)
                                     , pucBuf           := (#WrTaskInfo.Handshake)$^USINT
                                     ) <> SDIAS_OK then
          CyclicMsgMarker.PostIt.GetWrInfoFailed := TRUE;

        end_if;
        if SDIAS_iGetNodePropertyIndex(hNodeHandle      := udNodeHandle
                                     , udIndex          := 2
                                     , udPropertyId     := SDM_PROP_TASK_ERROR_INFO_FLAGS
                                     , pudPropertyValue := (#WrTaskInfo.ErrorInfoFlags)$^UDINT
                                     ) <> SDIAS_OK then
          CyclicMsgMarker.PostIt.GetWrInfoFailed := TRUE;
        end_if;
      end_if;

//**********************************************************************************************************************************************************
    _BUS_IF_POST_INIT_RT_READY:
      // if we got an error => return it
      if InitSSW = _ErrorOccured then
        ret_code := ERROR;

      // if we're not ready, return busy
      elsif RtSSW <> _Operational then
        ret_code := BUSY;
      end_if;

//**********************************************************************************************************************************************************
    CMD_GET_HW_TIMESTAMP:

      if RtSSW = _Operational then
        // SDIASManager gets Time every RtPreScan, no need to pass on the command
        ret_code := READY;

        pResult^.uiLng      := sizeof(t_GetHwTimestampResult);
        pResult^.aData[0]$t_GetHwTimestampResult.udVersion   := 1;
        pResult^.aData[0]$t_GetHwTimestampResult.uiTimeStamp := uiHWTimestamp;
      else
        // forward it to bus interface
        ret_code := ToBusInterface.NewInst(pPara, pResult);
      end_if;

//**********************************************************************************************************************************************************
    _BUS_IF_CREATE_MUTEX,
    _BUS_IF_SET_REQUIRED_ERROR,
    _BUS_IF_GET_BUSCYCLE_TIME,
    _BUS_IF_GET_DEACTIVATED_STATE,
    _BUS_IF_GET_HW_PATH,
    _BUS_IF_IS_VARAN_AVAILABLE,
    _BUS_IF_SET_RUN_STATE,
    _BUS_IF_SET_REQUIRED:
      // forward it to bus interface
      ret_code := ToBusInterface.NewInst(pPara, pResult);
//**********************************************************************************************************************************************************

//*****************************************************************************
//** COMMANDS FROM SDIAS MANAGER ITSELF                                      **
//*****************************************************************************

//**********************************************************************************************************************************************************
		SDIAS_CMD_SDO_RESPONSE:
      ret_code := ReceiveSDOResponse(Command:=pPara^.aPara[0]$t_SDIAS_SDO_Cmd,
                                     Offset:=pPara^.aPara[1]$HINT,
                                     Length:=pPara^.aPara[2]$USINT,
                                     Result:=pPara^.aPara[3]$iprStates,
                                     pResponseBuffer:=pPara^.aPara[4]$^USINT,
                                     ResponseLength:=pPara^.aPara[5]$USINT
                                     );

//**********************************************************************************************************************************************************
  else
    // unknown command
    if bUnknownCmdLogged = FALSE then
      bUnknownCmdLogged := TRUE;
#ifdef HWC_LogValue1
      HWC_LogValue1(this, "@006F (SdiasManager::ClassState::NewInst) [SL] Unknown command: 0x{0}", pPara^.uiCmd);
#endif
    end_if;

    ret_code := ERROR;
	END_CASE;

END_FUNCTION

FUNCTION SdiasManager::AddAccess
	VAR_INPUT
		AccessType 	: t_eAccessType;
		pThis 	: ^SdiasBase;
		Place 	: UDINT;
		Required 	: DINT;
		Offset 	: HINT;
		Length 	: UINT;
		ppData 	: pVoid;
		ppStateByte 	: pVoid;
		ppControlByte 	: pVoid;
		pAccessHandle 	: ^UDINT;
		WaitForAccessHandle 	: UDINT;
		bCtrlAcc0 	: BOOL;
	END_VAR
	VAR_OUTPUT
		Success 	: BOOL;
	END_VAR

  // check place
  if Place <= SDIAS_MAX_PLACE_NR then
    // check this pointer
    if pThis then
      // check other pointers as input parameters
      if ppData & ppStateByte & ppControlByte then
        // check offset and length for valid access
        if (Length > 0) & ((Offset + Length) <= SIZE_PER_SDIAS_CLIENT) then

          // remember the highest place to save time in module scanning operations like calling the realtime methods
          if (Place > MaxPlace) | (MaxPlace = SDIAS_PLACE_NO_MODULE_ADDED_SO_FAR) then
            MaxPlace := Place;
          end_if;

          // if it's a dynamic access on local SDIAS, check if the OS-Interface is available
          if ConnectionType = SDIAS_CON_LOCAL_uC then
            if ((AccessType = _ReadDynamic) | (AccessType = _WriteDynamic)) & (pSDIAS^.udVersion < SDIAS_CIL_VERSION_SUPPORTS_DYNAMIC_DO) then
#ifdef HWC_LogValue1
              HWC_LogValue1(this, "@0070 (SdiasManager::AddAccess) Newer OS Version needed for dynamic accesses on local SDIAS. Access for module at place 0x{0} can't be created!", Place);
#endif
              ModuleObjInfo[Place].pInitState^ := _UnknownCommand;
              InitError := _UnknownCommand;
              Success := FALSE;
              return;
            end_if;
          end_if;

          // remember the access
          Success := AddAccessToList(AccessType           := AccessType,
                                     Place                := Place,
                                     Offset               := Offset,
                                     Length               := Length,
                                     ppData               := ppData,
                                     ppStateByte          := ppStateByte,
                                     ppControlByte        := ppControlByte,
                                     pAccessHandle        := pAccessHandle,
                                     WaitForAccessHandle  := WaitForAccessHandle,
                                     bCtrlAcc0            := bCtrlAcc0,
                                     bIsFarAcc            := FALSE
                                     );

          // if adding failed classstate and initerrorstate are already set
          if Success = FALSE then
#ifdef HWC_LogValue1
            HWC_LogValue1(this, "@0071 (SdiasManager::AddAccess) Failed to add Access for Module at Place 0x{0}", Place);
#endif
          end_if;
        else  //add far memory access
          if (Length > 0) & (Length <= SDIAS_MAX_SIZE_FAR_MEM_ACCESS) & ((Offset + Length) > SIZE_PER_SDIAS_CLIENT) &
             ((Offset + Length) <= (SDIAS_1K_BLOCK_NO*SIZE_PER_SDIAS_CLIENT)) & (bCtrlAcc0 = FALSE) & FarMemoryAccessAvailable() then
            // remember the access
            Success := AddAccessToList(AccessType           := AccessType,
                                       Place                := Place,
                                       Offset               := Offset,
                                       Length               := Length,
                                       ppData               := ppData,
                                       ppStateByte          := ppStateByte,
                                       ppControlByte        := ppControlByte,
                                       pAccessHandle        := pAccessHandle,
                                       WaitForAccessHandle  := WaitForAccessHandle,
                                       bCtrlAcc0            := bCtrlAcc0,
                                       bIsFarAcc            := TRUE
                                       );

            // if adding failed classstate and initerrorstate are already set
            if Success = FALSE then
#ifdef HWC_LogValue1
              HWC_LogValue1(this, "@00DA (SdiasManager::AddAccess) Failed to add far memory access for Module at Place 0x{0}!", Place);
#endif

            end_if;
          else
#ifdef HWC_LogValue3
            HWC_LogValue3(this, "@0072 (SdiasManager::AddAccess) Invalid access for module at place: 0x{0}. Check offset (0x{1}) and length (0x{2})!", Place, Offset, Length);
#endif
            ModuleObjInfo[Place].pInitState^ := _DOLAddressInvalid;
            InitError := _DOLAddressInvalid;
            Success := FALSE;
          end_if;
        end_if;
      else
#ifdef HWC_LogValue1
        HWC_LogValue1(this, "@0073 (SdiasManager::AddAccess) Invalid pointer as input parameter for module at place: 0x{0}", Place);
#endif
        ModuleObjInfo[Place].pInitState^ := _MemoryFault;
        InitError := _MemoryFault;
        Success := FALSE;
      end_if;
    else
#ifdef HWC_LogValue1
      HWC_LogValue1(this, "@0074 (SdiasManager::AddAccess) Invalid this pointer for module at place: 0x{0}", Place);
#endif
      ModuleObjInfo[Place].pInitState^ := _MemoryFault;
      InitError := _MemoryFault;
      Success := FALSE;
    end_if;
  else
#ifdef HWC_LogValue2
    HWC_LogValue2(this, "@0075 (SdiasManager::AddAccess) Invalid Place number: 0x{0}. Maximum is 0x{1}", Place, SDIAS_MAX_PLACE_NR);
#endif
    if pThis then
      pThis^.ClassState := _InvalidDeviceAddress;
    end_if;
    InitError := _InvalidDeviceAddress;
    Success := FALSE;
  end_if;

  // if it was an access of a required module => required error
  if Required & (Success = FALSE) then
    SetRequiredError(pThis, Place);
  end_if;

END_FUNCTION

FUNCTION SdiasManager::ConnectEvent
  VAR
  	tempCmd         : CmdStruct;
    _result         : results;
    dataResetDO     : t_ResetDOCfg;
    Settings        : t_LoginSettings;
  END_VAR

  if b_PostInitFinished = FALSE then
    ConnectDuringPostInitCounter += 1;

    // don't reinit in postinit (ignore call from OS)
    if ConnectDuringPostInitCounter >= 2 then
      b_MultipleConnectInInit := TRUE;
      return;
    end_if;
  end_if;

  // install post init call back only if we're still in init (if we install it in init(), we may get called even the module is not connected)
  if us_Firstscan < 12 then
    tempCmd.uiCmd := _BUS_IF_WAIT_4_POST_INIT;
#pragma warning(disable: 74);
    Settings := 0;
#pragma warning(default: 74);
    Settings.Wait4DOCreation := MaxPlace <> SDIAS_PLACE_NO_MODULE_ADDED_SO_FAR;
    if Settings.Wait4DOCreation & (ConnectionType = SDIAS_CON_VIA_VARAN_uC) then
      Settings.Wait4MoveDOCreation := TRUE;
    end_if;
    Settings.Wait4SyncSend := TRUE;

    tempCmd.aPara[0] := Settings;
    ToBusInterface.NewInst(pPara:=#tempCmd, pResult:=#_result);

    if _result.aData[0]$t_BusIFRetvalErrorcode <> _BUS_IF_RETVAL_OK then
#ifdef HWC_LogError
      HWC_LogError(this, "@0076 (SdiasManager::ConnectEvent) Failed to install post init callback");
#endif
      InitError := _InvalidConfguration;
    end_if;
  else
    b_PostInitFinished := TRUE;
  end_if;

  if ConnectionType = SDIAS_CON_VIA_VARAN_uC then

    // reset data objects (calculate retry timeout)
    tempCmd.uiCmd     := _BUS_IF_RESET_DO;
    tempCmd.aPara[0]  := (#dataResetDO)$DINT;

    dataResetDO.Handle := ASYReadDO.Handle;

    ToBusInterface.NewInst(pPara:=#tempCmd, pResult:=#_result);
    if _result.aData[0]$t_BusIFRetvalErrorcode <> _BUS_IF_RETVAL_OK then
#ifdef HWC_LogError
      HWC_LogError(this, "@0077 (SdiasManager::ConnectEvent) Failed reset DO for the asynchronous read data");
#endif
    end_if;

    dataResetDO.Handle := ASYWriteDO.Handle;

    ToBusInterface.NewInst(pPara:=#tempCmd, pResult:=#_result);
    if _result.aData[0]$t_BusIFRetvalErrorcode <> _BUS_IF_RETVAL_OK then
#ifdef HWC_LogError
      HWC_LogError(this, "@0078 (SdiasManager::ConnectEvent) Failed reset DO for the asynchronous write data");
#endif
    end_if;
  end_if;

  if ConnectionType = SDIAS_CON_VIA_VARAN_uC then
    // set online server first on 1 if data is valid
    tempCmd.uiCmd    := _BUS_IF_SET_ONLINE;
    tempCmd.aPara[0] := 0;

    ToBusInterface.NewInst(pPara:=#tempCmd, pResult:=#_result);

    if _result.aData[0]$t_BusIFRetvalErrorcode <> _BUS_IF_RETVAL_OK then
#ifdef HWC_LogError
      HWC_LogError(this, "@0079 (SdiasManager::ConnectEvent) Failed to set Online server.");
#endif
    end_if;
  end_if;

  // reset max durations as it marks the first run
  WriteTaskInfo.MaxDuration := 0;
  ReadTaskInfo.MaxDuration := 0;

  InitSSW     := _StartInit;
  b_Ready4Rt  := FALSE;
  RtSSW       := _RtIdle;
  ClassState  := _NotInitialized;
  Online      := 1;

END_FUNCTION

FUNCTION SdiasManager::DisconnectEvent
  VAR
  	i : UDINT;
  END_VAR

  // if there is a required error, we would disguise it, if we call the disconnect interfaces
  if ClassState <> _RequiredError then

    // tell all the connected modules
    if MaxPlace <> SDIAS_PLACE_NO_MODULE_ADDED_SO_FAR then
      for i := 0 to MaxPlace do
        if ModuleObjInfo[i].pThis then
          ModuleObjInfo[i].pThis^.DisconnectEvent();
        end_if;
      end_for;
    end_if;

    ClassState := _NoHardware;

    FirmwareVersion := 0;
  end_if;

  Online := 0;

END_FUNCTION

FUNCTION SdiasManager::InterruptEvent

  // set only the state (we're in the interrupt and have to be fast)
  if b_IsRequired then
    ClassState := _HardwareRequiredIRQ;
  else
    ClassState := _HardwareNotRequiredIRQ;
  end_if;

  Online := 0;

END_FUNCTION

FUNCTION SdiasManager::SdiasManager
	VAR_OUTPUT
		ret_code 	: ConfStates;
	END_VAR

  ClassState := _NotInitialized;

#ifdef HWC_LogInit
  HWC_LogInit();
#else
  #pragma message("Warning! Log and trace messages of this class require a newer version of class HwControl. Please update for full functionality!")
#endif

  //get pointer for sdias function
	if OS_CILGET( INTERFACE_SDIAS, #pSDIAS ) then
#ifdef HWC_LogError
    HWC_LogError(this, "@007A (SdiasManager::SdiasManager) Failed to get SDIAS OS-Interface. A newer OS is necessary to use SDIAS");
#endif
  end_if;

  if (OS_CILGet("LSL_MULTITASK", #mt_api$void)) THEN
#ifdef HWC_LogError
    HWC_LogError(this, "@007B (SdiasManager::SdiasManager) Failed to get MULTITASK OS-Interface for Mutex usage");
#endif
  end_if;

  //Get pointer for pll interface for sync out settings
  OS_CILGet(INTERFACE_PLL, #pPLL$void); //No LogError because not every CPU has an PLL Interface

  MaxPlace := SDIAS_PLACE_NO_MODULE_ADDED_SO_FAR;

  //Set Supported Features of the sdias manager class
  SupportedFeatures.DefAcc4InitAcc := TRUE;

	ret_code := C_OK;

END_FUNCTION

FUNCTION SdiasManager::ChangeAsyRd
	VAR_INPUT
		Offset 	: HINT;
		Length 	: USINT;
		RunState 	: t_BusIFRunState;
		UsageType 	: t_AsyDOUsage;
	END_VAR
	VAR_OUTPUT
		Success 	: BOOL;
	END_VAR
  VAR
    dataUPDATEDO    : t_UpdateDOCfg;
  	tempCmd         : CmdStruct;
    _result         : results;
    dataSETRUNSTATE : t_SetRunStateCfg;
  END_VAR

  if (AsyReadUsage = _NotUsed) | (AsyReadUsage = UsageType) then

    // if length = zero we may just want to stop the DO
    if Length then
      ASYReadDO.Offset := Offset;
      ASYReadDO.Length := Length;

      dataUPDATEDO.Handle               := ASYReadDO.Handle;
      dataUPDATEDO.ud_addressoff_read   := ASYReadDO.Offset;
      dataUPDATEDO.ud_length_read       := ASYReadDO.Length;

      tempCmd.uiCmd         := _BUS_IF_UPDATE_DO;
      tempCmd.aPara[0]      := (#dataUPDATEDO)$DINT;

      ToBusInterface.NewInst(pPara:=#tempCmd, pResult:=#_result);
      if _result.aData[0]$t_BusIFRetvalErrorcode <> _BUS_IF_RETVAL_OK then
#ifdef HWC_LogError
        HWC_LogError(this, "@007C (SdiasManager::ChangeAsyRd) Failed to change asynchron read access");
#endif
      end_if;
    end_if;

    // set runstate
    dataSETRUNSTATE.Handle      := ASYReadDO.Handle;
    dataSETRUNSTATE.NewRunState := RunState;

    tempCmd.uiCmd         := _BUS_IF_SET_RUN_STATE;
    tempCmd.aPara[0]      := (#dataSETRUNSTATE)$DINT;

    ToBusInterface.NewInst(pPara:=#tempCmd, pResult:=#_result);

    if _result.aData[0]$t_BusIFRetvalErrorcode <> _BUS_IF_RETVAL_OK then
#ifdef HWC_LogError
      HWC_LogError(this, "@007D (SdiasManager::ChangeAsyRd) Error changing the run state of the asynchron read access!");
#endif
    end_if;

    if RunState = _BUS_IF_RUN_STATE_NO_RUN then
      AsyReadUsage := _NotUsed;
    else
      AsyReadUsage := UsageType;
    end_if;

    Success := TRUE;
  else
#ifdef HWC_LogError
    HWC_LogError(this, "@007E (SdiasManager::ChangeAsyRd) Failed to use DO (already in use by another task)");
#endif
    Success := FALSE;
  end_if;

END_FUNCTION

FUNCTION SdiasManager::ChangeAsyWr
	VAR_INPUT
		Offset 	: HINT;
		Length 	: USINT;
		RunState 	: t_BusIFRunState;
		UsageType 	: t_AsyDOUsage;
	END_VAR
	VAR_OUTPUT
		Success 	: BOOL;
	END_VAR
  VAR
    dataUPDATEDO    : t_UpdateDOCfg;
  	tempCmd         : CmdStruct;
    _result         : results;
    dataSETRUNSTATE : t_SetRunStateCfg;
  END_VAR

  if (AsyWriteUsage = _NotUsed) | (AsyWriteUsage = UsageType) then
    // if a watchdog trigger has to be sent, ignore other requests
    if b_SendWdTrigger & (UsageType <> _UsedByWD) then
      AsyWriteUsage := _UsedByWD;
      Success := FALSE;
      return;
    end_if;

    // if length = zero we may just want to stop the DO
    if Length then
      ASYWriteDO.Offset := Offset;
      ASYWriteDO.Length := Length;

      dataUPDATEDO.Handle               := ASYWriteDO.Handle;
      dataUPDATEDO.ud_addressoff_write  := ASYWriteDO.Offset;
      dataUPDATEDO.ud_length_write      := ASYWriteDO.Length;

      tempCmd.uiCmd         := _BUS_IF_UPDATE_DO;
      tempCmd.aPara[0]      := (#dataUPDATEDO)$DINT;

      ToBusInterface.NewInst(pPara:=#tempCmd, pResult:=#_result);
      if _result.aData[0]$t_BusIFRetvalErrorcode <> _BUS_IF_RETVAL_OK then
#ifdef HWC_LogError
        HWC_LogError(this, "@007F (SdiasManager::ChangeAsyWr) Failed to change asynchron write access");
#endif
      end_if;
    end_if;

    // set runstate
    dataSETRUNSTATE.Handle      := ASYWriteDO.Handle;
    dataSETRUNSTATE.NewRunState := RunState;

    tempCmd.uiCmd         := _BUS_IF_SET_RUN_STATE;
    tempCmd.aPara[0]      := (#dataSETRUNSTATE)$DINT;

    ToBusInterface.NewInst(pPara:=#tempCmd, pResult:=#_result);

    if _result.aData[0]$t_BusIFRetvalErrorcode <> _BUS_IF_RETVAL_OK then
#ifdef HWC_LogError
      HWC_LogError(this, "@0080 (SdiasManager::ChangeAsyWr) Error changing the run state of the asynchron write access!");
#endif
    end_if;

    if RunState = _BUS_IF_RUN_STATE_NO_RUN then
      AsyWriteUsage := _NotUsed;
    else
      AsyWriteUsage := UsageType;
    end_if;

    Success := TRUE;
  else
    // only print the message if there is no collision with watchdog (collision with watchdog is very likely)
    if (AsyWriteUsage <> _UsedByWD) & (UsageType <> _UsedByWD) then
#ifdef HWC_LogError
      HWC_LogError(this, "@0081 (SdiasManager::ChangeAsyWr) Failed to use DO (already in use by another task)");
#endif
    end_if;

    Success := FALSE;
  end_if;

END_FUNCTION

FUNCTION SdiasManager::AddAccessToList
	VAR_INPUT
		AccessType 	: t_eAccessType;
		Place 	: UDINT;
		Offset 	: HINT;
		Length 	: UINT;
		ppData 	: pVoid;
		ppStateByte 	: pVoid;
		ppControlByte 	: pVoid;
		pAccessHandle 	: ^UDINT;
		WaitForAccessHandle 	: UDINT;
		bCtrlAcc0 	: BOOL;
		bIsFarAcc 	: BOOL;
	END_VAR
	VAR_OUTPUT
		Success 	: BOOL;
	END_VAR
  VAR
    pHelpAccess : ^t_AccessElement;
  END_VAR

  if ModuleObjInfo[Place].pFirstAccess = NIL then
    ModuleObjInfo[Place].pFirstAccess$pVoid := ToStdLib.Malloc(size:=sizeof(t_AccessElement));
    pHelpAccess := ModuleObjInfo[Place].pFirstAccess;
  else
    pHelpAccess := ModuleObjInfo[Place].pFirstAccess;
    while pHelpAccess^.pNext <> NIL do
      pHelpAccess := pHelpAccess^.pNext;
    end_while;
    pHelpAccess^.pNext$pVoid := ToStdLib.Malloc(size:=sizeof(t_AccessElement));
    pHelpAccess := pHelpAccess^.pNext;
  end_if;

  if pHelpAccess <> NIL then
    pHelpAccess^.eAccessType                  := AccessType;
    pHelpAccess^.usPlace                      := Place$USINT;
    pHelpAccess^.hiOffset                     := Offset;
    pHelpAccess^.uiLength                     := Length;
    pHelpAccess^.ppData                       := ppData;
    pHelpAccess^.ppStateByte                  := ppStateByte$^t_SDIAS_pStateByte;
    pHelpAccess^.ppControlByte                := ppControlByte$^t_SDIAS_pControlByte;
    pHelpAccess^.pWaitForAccess               := WaitForAccessHandle$^t_AccessElement;
    pHelpAccess^.udOSDOHandle                 := NIL;
    pHelpAccess^.pNext                        := NIL;
    pHelpAccess^.bCtrlAcc0                    := bCtrlAcc0;
    pHelpAccess^.bIsFarAcc                    := bIsFarAcc;

    // count the data for the varan payload frames
    case AccessType of
      _Read:
          ISOWriteDO.Length += sizeof(t_SDIAS_ControlByte); // control byte
          ISOReadDO.Length  += sizeof(t_SDIAS_StateByte) + Length; // state byte + data length

      _Write:
          ISOWriteDO.Length += sizeof(t_SDIAS_ControlByte) + Length; // control byte + data length
          ISOReadDO.Length  += sizeof(t_SDIAS_StateByte); // state byte;

      _ReadDynamic:
          ISOWriteDO.Length += sizeof(t_SDIAS_ControlStructDynamic); // control byte + length info + offset info
          ISOReadDO.Length  += sizeof(t_SDIAS_StateByte) + Length; // state byte + data length

      _WriteDynamic:
          ISOWriteDO.Length += sizeof(t_SDIAS_ControlStructDynamic) + Length; // control byte + length info + offset info + data length
          ISOReadDO.Length  += sizeof(t_SDIAS_StateByte); // state byte;
    end_case;

    // only for easier debugging
    ModuleObjInfo[Place].AccessNo += 1;

    if pAccessHandle then
      pAccessHandle^ := pHelpAccess$UDINT;
    end_if;

    Success := TRUE;
  else
    ClassState := _MemoryFault;
    InitError := _MemoryFault;
#ifdef HWC_LogError
    HWC_LogError(this, "@0082 (SdiasManager::AddAccessToList) Failed to allocate memory for an SDIAS Access");
#endif

    if pAccessHandle then
      pAccessHandle^ := 0;
    end_if;

    Success := FALSE;
  end_if;

END_FUNCTION

FUNCTION SdiasManager::AddBroadCastAccessesToList
  VAR
    i : USINT;
  END_VAR

  // Memory for Access data is already held by SDIAS Manager, No need for pHelpAccess

  // count the data for the varan payload frames
  // Access type is control broadcast 2 Byte, Read 0 Byte
  if SupportedFeatures.TimeBroadCastSupported then
    for i := 0 to SDIAS_NR_TIMEBROADCAST_DOS - 1 do
      ISOWriteDO.Length += sizeof(t_SDIAS_ControlByte) + sizeof(UINT);  // control byte + data length
      ISOReadDO.Length  += sizeof(t_SDIAS_StateByte);                   // state byte
    end_for;
  end_if;

END_FUNCTION

FUNCTION SdiasManager::CheckTimeBroadCastSupported
	VAR_OUTPUT
		bTimeBroadCastSupported 	: BOOL;
	END_VAR
  VAR
    tempCmd             : CmdStruct;
    _result             : results;
    retval              : iprStates;
  END_VAR

  // Countercheck
  bTimeBroadCastSupported := TRUE;

  // Check if broadcast command is supported by OS
  if ConnectionType = SDIAS_CON_LOCAL_uC then

    // OS is only needed for local SDIAS
    if (pSDIAS^.udVersion < SDIAS_CILVERSION_BROADCAST) then
      bTimeBroadCastSupported := FALSE;
    end_if;

  end_if;

  // Check if broadcast command is supported SDIAS Manager
  if FeatureInfo.ProtocolVersion < SDIAS_PROTOCOLVERSION_BROADCAST then
    bTimeBroadCastSupported := FALSE;
  end_if;

  // Timestamp of HWControl must be valid
  tempCmd.uiCmd := CMD_GET_HW_TIMESTAMP;
  tempCmd.aPara[0]$t_GetHwTimestampCmd.udVersion    := 1;
  tempCmd.aPara[0]$t_GetHwTimestampCmd.udCoreSelect := 0;

  _result.aData[0]$t_GetHwTimestampResult.udVersion := 0; // Init return Value incase command is not implemented in HWControl

  retval := ToBusInterface.NewInst(#tempCmd, #_result);

  if retval <> READY then
    bTimeBroadCastSupported := FALSE;
  elsif _result.aData[0]$t_GetHwTimestampResult.udVersion < 1 then
    bTimeBroadCastSupported := FALSE;
  end_if;

END_FUNCTION

FUNCTION VIRTUAL SdiasManager::ReceiveSDOResponse
	VAR_INPUT
		Command 	: t_SDIAS_SDO_Cmd;
		Offset 	: HINT;
		Length 	: USINT;
		Result 	: iprStates;
		pResponseBuffer 	: ^USINT;
		ResponseLength 	: USINT;
	END_VAR
	VAR_OUTPUT
		ret_code 	: iprStates;
	END_VAR

  ret_code := READY;

  case Command of
    SDIAS_SDO_CMD_REBUILD_SDIAS:
      // if it succeeded, check if we have something to do
      if Result = READY then
        // everthing is fine
      else
        // an error occured while performing the operation
#ifdef HWC_LogError
        HWC_LogError(this, "@0083 (SdiasManager::ReceiveSDOResponse) Rebuild SDIAS SDO command failed!");
#endif
      end_if;
    SDIAS_SDO_CMD_SET_NEW_END:
      // if it succeeded, check if we have something to do
      if Result = READY then
        // everthing is fine
        bReceivedNewEndRsp := TRUE;
      else
        // an error occured while performing the operation
#ifdef HWC_LogError
        HWC_LogError(this, "@0084 (SdiasManager::ReceiveSDOResponse) Set new DOL end command failed!");
#endif
      end_if;

  else
    ret_code := ERROR;
#ifdef HWC_LogError
    HWC_LogError(this, "@0085 (SdiasManager::ReceiveSDOResponse) Invalid command in SDO response!");
#endif
  end_case;

END_FUNCTION

FUNCTION SdiasManager::AddSDOReq
	VAR_INPUT
		pCmdSvr 	: ^SvrChCmd;
		Command 	: t_SDIAS_SDO_Cmd;
		Place 	: USINT;
		CmdLength 	: USINT;
		pReqBuf 	: ^USINT;
	END_VAR
	VAR_OUTPUT
		sd_retval 	: DINT;
	END_VAR

  // protect via mutex because this can be called from different task priorities
  OS_MT_WAIT(pv_Mutex);

  // if the buffer is full, or the next element in the buffer is already in use
  if (SDOHandling.pWrite^.Command <> SDIAS_SDO_CMD_INVALID) then
    sd_retval := SDIAS_MAILBOX_FULL;
    OS_MT_SIGNAL(pv_Mutex);
    return;
  end_if;

  // check the pointer first (if needed)
  if CmdLength then
    if pReqBuf then
      _memcpy(ptr1:=#SDOHandling.pWrite^.ReqBufData, ptr2:=pReqBuf, cntr:=CmdLength);
    else
      sd_retval := SDIAS_INVALID_PARAM_DATA_BUFFER;
      OS_MT_SIGNAL(pv_Mutex);
      return;
    end_if;
  end_if;

  SDOHandling.pWrite^.pCallBackSvr := pCmdSvr;
  SDOHandling.pWrite^.NMTCommand := 0;
  SDOHandling.pWrite^.SDIASPlace := Place;
  SDOHandling.pWrite^.CmdLength := CmdLength;

  case Command of
    SDIAS_SDO_CMD_MEM_READ,
    SDIAS_SDO_CMD_MEM_WRITE,
    SDIAS_SDO_CMD_CTRL_READ,
    SDIAS_SDO_CMD_CTRL_WRITE:
//    SDIAS_SDO_CMD_SPI_READ,
//    SDIAS_SDO_CMD_SPI_WRITE:
      // store offset and length for read and write accesses
      SDOHandling.pWrite^.RdWrHead := pReqBuf^$t_SDIAS_SDO_RdWr_Head;
    SDIAS_SDO_CMD_SPI_READ,
    SDIAS_SDO_CMD_SPI_WRITE:

      // store offset and length for read and write accesses
      SDOHandling.pWrite^.RdWrHead := pReqBuf^$t_SDIAS_SDO_RdWr_Head;

  end_case;

  // command is the last thing to store, because it indicates a complete entry
  SDOHandling.pWrite^.Command := Command;

  // we increment our used entries in the buffer (only for debugging)
  SDOHandling.EntriesUsed     += 1;

  // after we successfully added this SDO, set the write pointer to the next element
  if SDOHandling.pWrite = SDOHandling.pLastEntry then
    SDOHandling.pWrite := SDOHandling.pRingBufMemStart;
  else
    SDOHandling.pWrite += sizeof(t_SDORingBufEntry);
  end_if;

  sd_retval := SDIAS_OK;

  OS_MT_SIGNAL(pv_Mutex);

END_FUNCTION

FUNCTION SdiasManager::CyclicSDOHandling
  VAR
  	i,j           : USINT;
    FoundIt       : BOOL;
		Offset 	      : HINT;
		Length 	      : USINT;
    pTempChannel  : ^t_SDOChannel;
    TempChannel   : t_SDOChannel;
    pRingBufEntry : ^t_SDORingBufEntry;
    FirstFound    : USINT;
    LastFound     : USINT;
    Channels2Add  : DINT;
    StartIndex    : USINT;
    EndIndex      : USINT;
    pCmdSvr       : ^SvrChCmd;
  	tempCmd       : CmdStruct;
    _result       : results;
    ReceiveBuffer : ARRAY [0..127] OF USINT;
    ReceiveLength : UDINT;
    sd_retval     : DINT;
    TempUDINT     : UDINT;
    OldChannelNo  : USINT;
  END_VAR

  // protect via mutex because this can be called from different task priorities
  OS_MT_WAIT(pv_Mutex);

  if ConnectionType = SDIAS_CON_VIA_VARAN_uC then

    // check sdo response first. if a channel is ready it can be used for the next request

    // GET SDO RESPONSE
    if (AsyReadUsage = _NotUsed) | (AsyReadUsage = _UsedBySDO) then

      // if the AsyRdDO is used for polling, we check if we got a response
      if AsyReadUsage = _UsedBySDO then
        StartIndex := ((ASYReadDO.Offset - SDOHandling.OffsetSDOResp) / sizeof(t_SDOChannel))$USINT;
        EndIndex := StartIndex + (ASYReadDO.Length / sizeof(t_SDOChannel))$USINT - 1;
        Offset := 0;
        for i := StartIndex to EndIndex do
          if SDOHandling.aChannelData[i].WaitForResponse then
            // check for the response (copy only header first)
            _memcpy(ptr1:=#TempChannel, ptr2:=ASYReadDO.pData$^t_SDOChannel + Offset, cntr:=sizeof(t_SDOChannel) - sizeof(t_SDOChannel.Data));
            pRingBufEntry := SDOHandling.aChannelData[i].pActElement;

            // if the header info is mirrored, the SDO is ready
            if ((TempChannel.MessageCounter AND SDIAS_MASK_MESSAGE_COUNTER) = pRingBufEntry^.MessageCounter) &
               (TempChannel.SDIASPlace = pRingBufEntry^.SDIASPlace) &
               (TempChannel.Command$t_SDIAS_SDO_Cmd = pRingBufEntry^.Command) then
